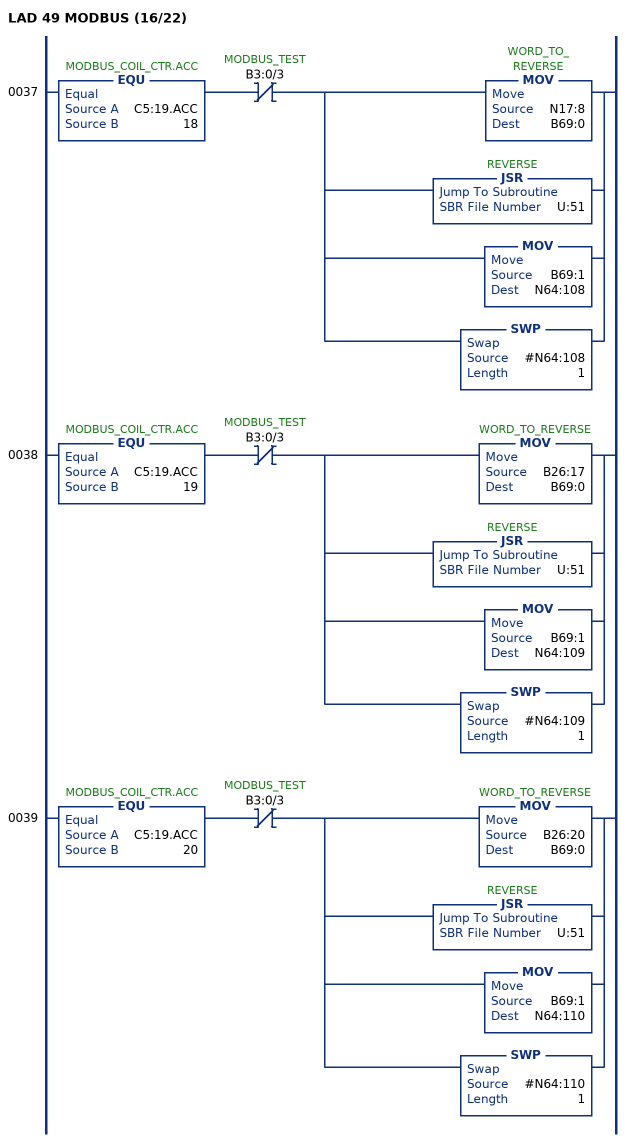
% Rung: 37 %
SOR EQU C5:19.ACC 18 XIO B3:0/3 BST MOV N17:8 B69:0 NXB JSR U:51 NXB MOV B69:1 N64:108 NXB SWP #N64:108 1 BND EOR
%   C5:19  MODBUS_COIL_CTR %
%   B3:0/3  MODBUS_TEST %
%   N17:8  ADS_B_PURIFY_WARNS  "WARNING ADS B Warnings" %
%   B69:0  WORD_TO_REVERSE %
%   U:51  REVERSE %
%   B69:1  REVERSED_WORD %
% Rung: 38 %
SOR EQU C5:19.ACC 19 XIO B3:0/3 BST MOV B26:17 B69:0 NXB JSR U:51 NXB MOV B69:1 N64:109 NXB SWP #N64:109 1 BND EOR
%   C5:19  MODBUS_COIL_CTR %
%   B3:0/3  MODBUS_TEST %
%   B26:17  GETTER_1_ALARMS %
%   B69:0  WORD_TO_REVERSE %
%   U:51  REVERSE %
%   B69:1  REVERSED_WORD %
% Rung: 39 %
SOR EQU C5:19.ACC 20 XIO B3:0/3 BST MOV B26:20 B69:0 NXB JSR U:51 NXB MOV B69:1 N64:110 NXB SWP #N64:110 1 BND EOR
%   C5:19  MODBUS_COIL_CTR %
%   B3:0/3  MODBUS_TEST %
%   B26:20  GET_1_OPEN_TC_ALARMS %
%   B69:0  WORD_TO_REVERSE %
%   U:51  REVERSE %
%   B69:1  REVERSED_WORD %

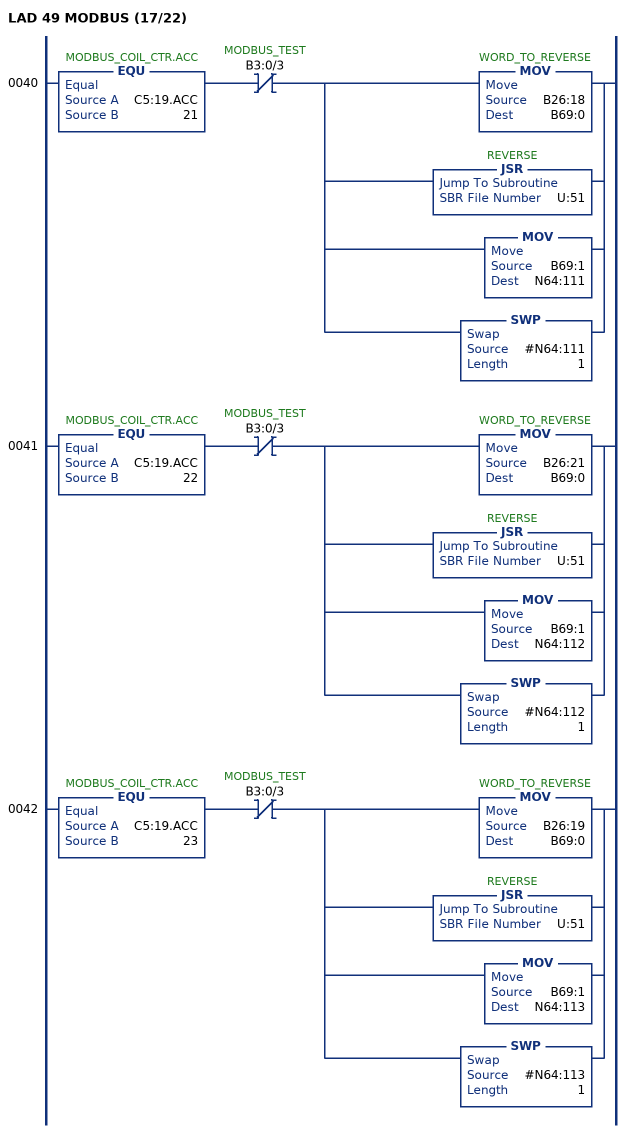
% Rung: 40 %
SOR EQU C5:19.ACC 21 XIO B3:0/3 BST MOV B26:18 B69:0 NXB JSR U:51 NXB MOV B69:1 N64:111 NXB SWP #N64:111 1 BND EOR
%   C5:19  MODBUS_COIL_CTR %
%   B3:0/3  MODBUS_TEST %
%   B26:18  GETTER_2_ALARMS %
%   B69:0  WORD_TO_REVERSE %
%   U:51  REVERSE %
%   B69:1  REVERSED_WORD %
% Rung: 41 %
SOR EQU C5:19.ACC 22 XIO B3:0/3 BST MOV B26:21 B69:0 NXB JSR U:51 NXB MOV B69:1 N64:112 NXB SWP #N64:112 1 BND EOR
%   C5:19  MODBUS_COIL_CTR %
%   B3:0/3  MODBUS_TEST %
%   B26:21  GET_2_OPEN_TC_ALARMS %
%   B69:0  WORD_TO_REVERSE %
%   U:51  REVERSE %
%   B69:1  REVERSED_WORD %
% Rung: 42 %
SOR EQU C5:19.ACC 23 XIO B3:0/3 BST MOV B26:19 B69:0 NXB JSR U:51 NXB MOV B69:1 N64:113 NXB SWP #N64:113 1 BND EOR
%   C5:19  MODBUS_COIL_CTR %
%   B3:0/3  MODBUS_TEST %
%   B26:19  GETTER_3_ALARMS %
%   B69:0  WORD_TO_REVERSE %
%   U:51  REVERSE %
%   B69:1  REVERSED_WORD %

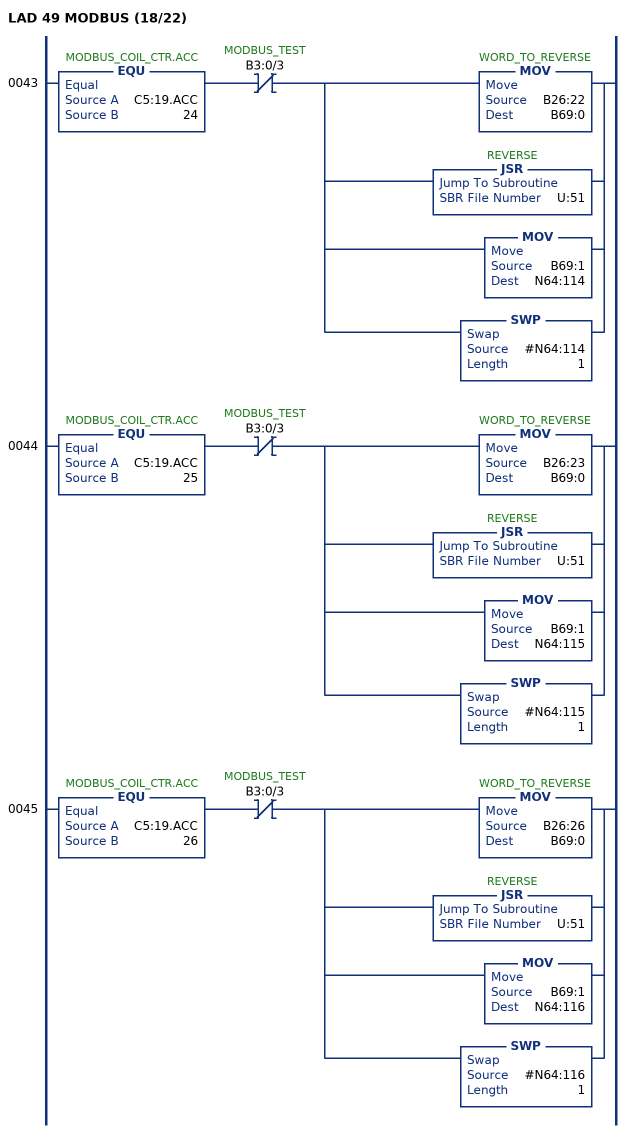
% Rung: 43 %
SOR EQU C5:19.ACC 24 XIO B3:0/3 BST MOV B26:22 B69:0 NXB JSR U:51 NXB MOV B69:1 N64:114 NXB SWP #N64:114 1 BND EOR
%   C5:19  MODBUS_COIL_CTR %
%   B3:0/3  MODBUS_TEST %
%   B26:22  GET_3_OPEN_TC_ALARMS %
%   B69:0  WORD_TO_REVERSE %
%   U:51  REVERSE %
%   B69:1  REVERSED_WORD %
% Rung: 44 %
SOR EQU C5:19.ACC 25 XIO B3:0/3 BST MOV B26:23 B69:0 NXB JSR U:51 NXB MOV B69:1 N64:115 NXB SWP #N64:115 1 BND EOR
%   C5:19  MODBUS_COIL_CTR %
%   B3:0/3  MODBUS_TEST %
%   B26:23  GETTER_1_WARNINGS %
%   B69:0  WORD_TO_REVERSE %
%   U:51  REVERSE %
%   B69:1  REVERSED_WORD %
% Rung: 45 %
SOR EQU C5:19.ACC 26 XIO B3:0/3 BST MOV B26:26 B69:0 NXB JSR U:51 NXB MOV B69:1 N64:116 NXB SWP #N64:116 1 BND EOR
%   C5:19  MODBUS_COIL_CTR %
%   B3:0/3  MODBUS_TEST %
%   B26:26  GET_1_OPEN_TC_WARNS %
%   B69:0  WORD_TO_REVERSE %
%   U:51  REVERSE %
%   B69:1  REVERSED_WORD %

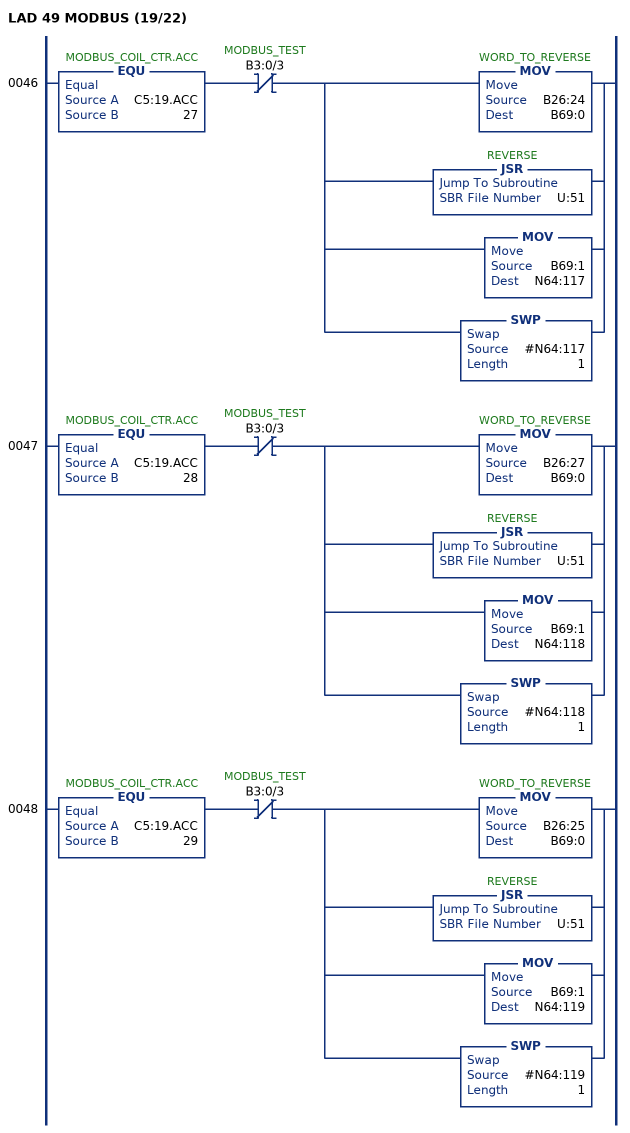
% Rung: 46 %
SOR EQU C5:19.ACC 27 XIO B3:0/3 BST MOV B26:24 B69:0 NXB JSR U:51 NXB MOV B69:1 N64:117 NXB SWP #N64:117 1 BND EOR
%   C5:19  MODBUS_COIL_CTR %
%   B3:0/3  MODBUS_TEST %
%   B26:24  GETTER_2_WARNINGS %
%   B69:0  WORD_TO_REVERSE %
%   U:51  REVERSE %
%   B69:1  REVERSED_WORD %
% Rung: 47 %
SOR EQU C5:19.ACC 28 XIO B3:0/3 BST MOV B26:27 B69:0 NXB JSR U:51 NXB MOV B69:1 N64:118 NXB SWP #N64:118 1 BND EOR
%   C5:19  MODBUS_COIL_CTR %
%   B3:0/3  MODBUS_TEST %
%   B26:27  GET_2_OPEN_TC_WARNS %
%   B69:0  WORD_TO_REVERSE %
%   U:51  REVERSE %
%   B69:1  REVERSED_WORD %
% Rung: 48 %
SOR EQU C5:19.ACC 29 XIO B3:0/3 BST MOV B26:25 B69:0 NXB JSR U:51 NXB MOV B69:1 N64:119 NXB SWP #N64:119 1 BND EOR
%   C5:19  MODBUS_COIL_CTR %
%   B3:0/3  MODBUS_TEST %
%   B26:25  GETTER_3_WARNINGS %
%   B69:0  WORD_TO_REVERSE %
%   U:51  REVERSE %
%   B69:1  REVERSED_WORD %

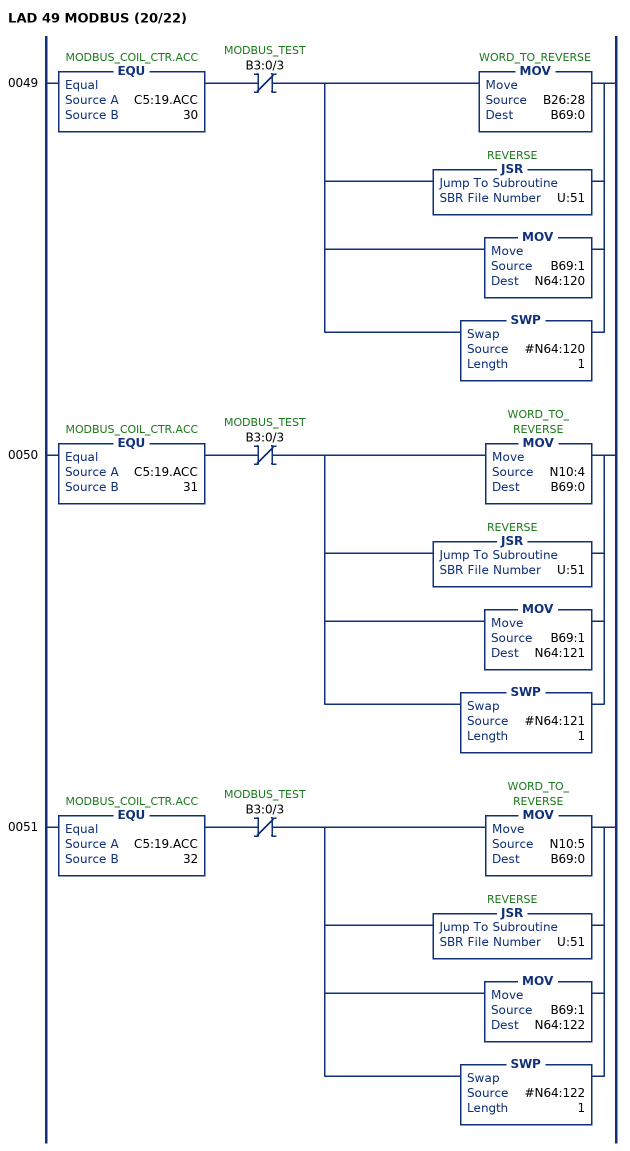
% Rung: 49 %
SOR EQU C5:19.ACC 30 XIO B3:0/3 BST MOV B26:28 B69:0 NXB JSR U:51 NXB MOV B69:1 N64:120 NXB SWP #N64:120 1 BND EOR
%   C5:19  MODBUS_COIL_CTR %
%   B3:0/3  MODBUS_TEST %
%   B26:28  GET_3_OPEN_TC_WARNS %
%   B69:0  WORD_TO_REVERSE %
%   U:51  REVERSE %
%   B69:1  REVERSED_WORD %
% Rung: 50 %
SOR EQU C5:19.ACC 31 XIO B3:0/3 BST MOV N10:4 B69:0 NXB JSR U:51 NXB MOV B69:1 N64:121 NXB SWP #N64:121 1 BND EOR
%   C5:19  MODBUS_COIL_CTR %
%   B3:0/3  MODBUS_TEST %
%   N10:4  H2_ALARMS %
%   B69:0  WORD_TO_REVERSE %
%   U:51  REVERSE %
%   B69:1  REVERSED_WORD %
% Rung: 51 %
SOR EQU C5:19.ACC 32 XIO B3:0/3 BST MOV N10:5 B69:0 NXB JSR U:51 NXB MOV B69:1 N64:122 NXB SWP #N64:122 1 BND EOR
%   C5:19  MODBUS_COIL_CTR %
%   B3:0/3  MODBUS_TEST %
%   N10:5  H2_WARNINGS %
%   B69:0  WORD_TO_REVERSE %
%   U:51  REVERSE %
%   B69:1  REVERSED_WORD %

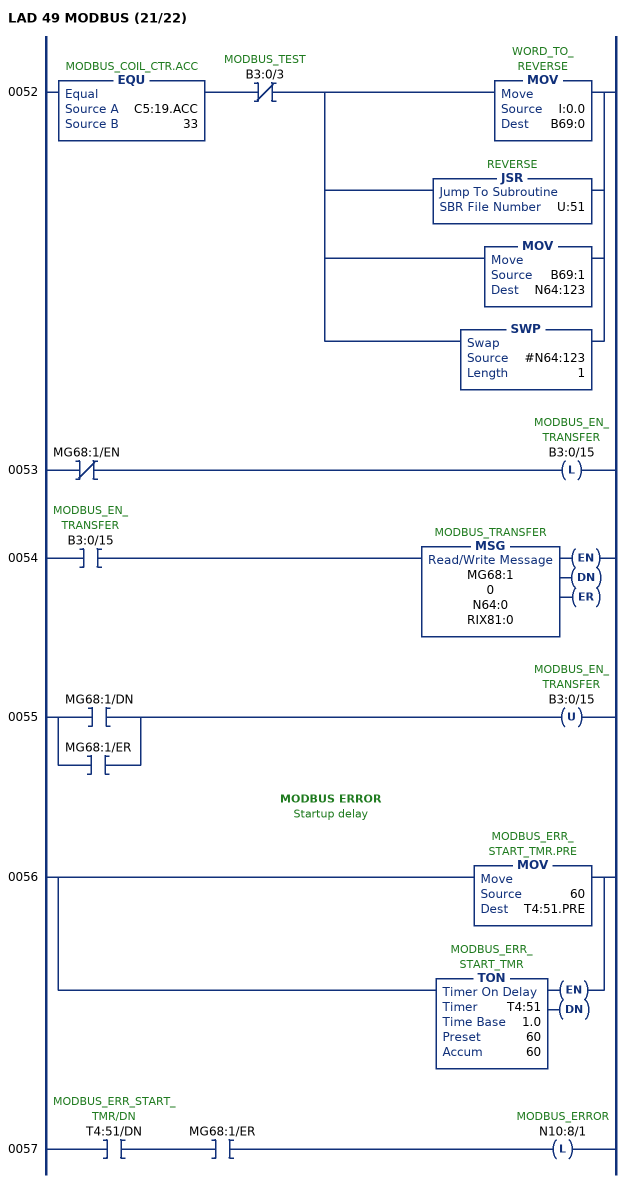
% Rung: 52 %
SOR EQU C5:19.ACC 33 XIO B3:0/3 BST MOV I:0.0 B69:0 NXB JSR U:51 NXB MOV B69:1 N64:123 NXB SWP #N64:123 1 BND EOR
%   C5:19  MODBUS_COIL_CTR %
%   B3:0/3  MODBUS_TEST %
%   B69:0  WORD_TO_REVERSE %
%   U:51  REVERSE %
%   B69:1  REVERSED_WORD %
% Rung: 53 %
SOR XIO MG68:1/EN OTL B3:0/15 EOR
%   B3:0/15  MODBUS_EN_TRANSFER %
% Rung: 54 %
SOR XIC B3:0/15 MSG MG68:1 0 N64:0 RIX81:0 EOR
%   B3:0/15  MODBUS_EN_TRANSFER %
%   MSG set-up: CIP Generic | 33 | 0 | ? | 0 | 0 | 0 | 0 | 172.16.14.73 | 0 | 0 | 172.16.14.73 | RIX81:0 | 10 | 4 | 150 | 3 | 4 | 96 | 3 | 252 | N64:0 %
%   MG68:1  MODBUS_TRANSFER %
%   N64:0  REGISTER_START %
% Rung: 55 %
SOR BST XIC MG68:1/DN NXB XIC MG68:1/ER BND OTU B3:0/15 EOR
%   B3:0/15  MODBUS_EN_TRANSFER %
% Rung: 56 %
% TITLE: MODBUS ERROR %
% Startup delay %
SOR BST MOV 60 T4:51.PRE NXB TON T4:51 1.0 60 60 BND EOR
%   T4:51  MODBUS_ERR_START_TMR %
% Rung: 57 %
SOR XIC T4:51/DN XIC MG68:1/ER OTL N10:8/1 EOR
%   T4:51  MODBUS_ERR_START_TMR %
%   N10:8/1  MODBUS_ERROR %

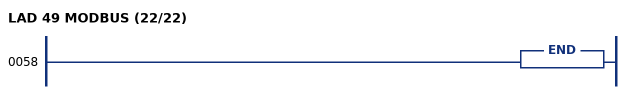
% Rung: 58 %
SOR END EOR

LADDER 50 "PLC FAULT"
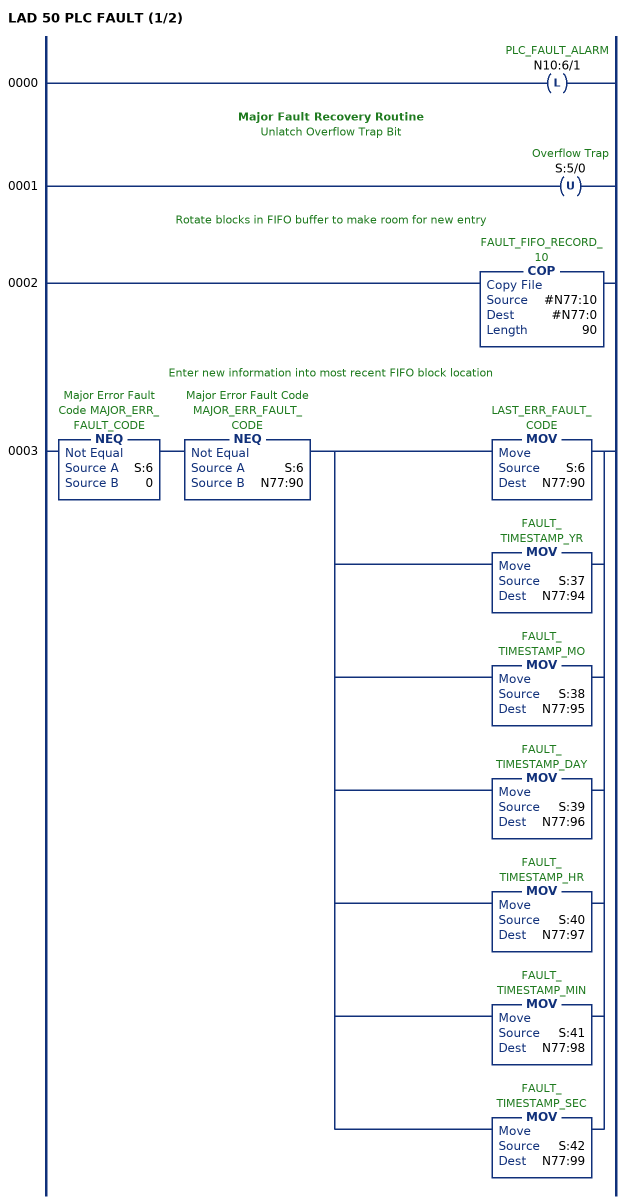
% Rung: 0 %
SOR OTL N10:6/1 EOR
%   N10:6/1  PLC_FAULT_ALARM %
% Rung: 1 %
% TITLE: Major Fault Recovery Routine %
% Unlatch Overflow Trap Bit %
SOR OTU S:5/0 EOR
%   S:5/0  "Overflow Trap" %
% Rung: 2 %
% Rotate blocks in FIFO buffer to make room for new entry %
SOR COP #N77:10 #N77:0 90 EOR
%   N77:10  FAULT_FIFO_RECORD_9 %
%   N77:0  FAULT_FIFO_RECORD_10 %
% Rung: 3 %
% Enter new information into most recent FIFO block location %
SOR NEQ S:6 0 NEQ S:6 N77:90 BST MOV S:6 N77:90 NXB MOV S:37 N77:94 NXB MOV S:38 N77:95 NXB MOV S:39 N77:96 NXB MOV S:40 N77:97 NXB MOV S:41 N77:98 NXB MOV S:42 N77:99 BND EOR
%   S:6  MAJOR_ERR_FAULT_CODE  "Major Error Fault Code" %
%   N77:90  LAST_ERR_FAULT_CODE %
%   S:37  RTC_YEAR  "Clock Calendar Year" %
%   N77:94  FAULT_TIMESTAMP_YR %
%   S:38  RTC_MONTH  "Clock Calendar Month" %
%   N77:95  FAULT_TIMESTAMP_MO %
%   S:39  RTC_DAY_OF_MONTH  "Clock Calendar Day" %
%   N77:96  FAULT_TIMESTAMP_DAY %
%   S:40  RTC_HOUR  "Clock Calendar Hours" %
%   N77:97  FAULT_TIMESTAMP_HR %
%   S:41  RTC_MINUTE  "Clock Calendar Minutes" %
%   N77:98  FAULT_TIMESTAMP_MIN %
%   S:42  RTC_SECOND  "Clock Calendar Seconds" %
%   N77:99  FAULT_TIMESTAMP_SEC %

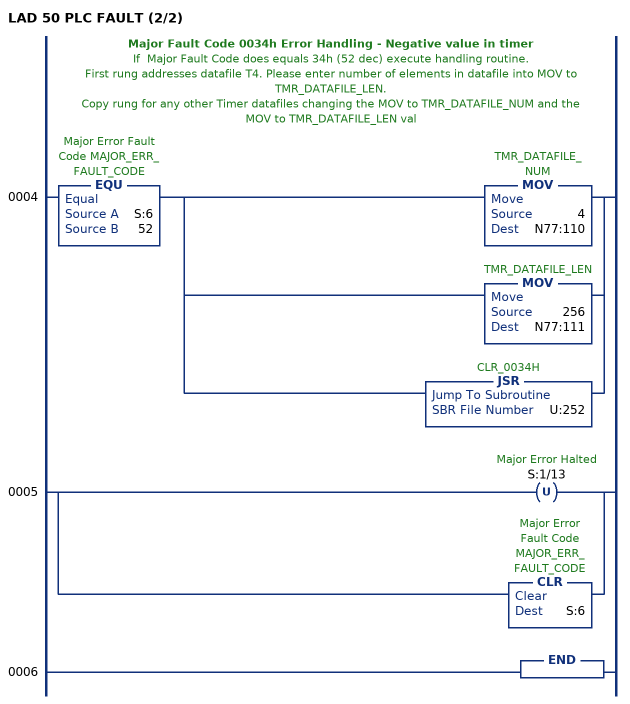
% Rung: 4 %
% TITLE: Major Fault Code 0034h Error Handling - Negative value in timer %
% If  Major Fault Code does equals 34h (52 dec) execute handling routine.
% First rung addresses datafile T4. Please enter number of elements in datafile into MOV to TMR_DATAFILE_LEN.
% Copy rung for any other Timer datafiles changing the MOV to TMR_DATAFILE_NUM and the MOV to TMR_DATAFILE_LEN val %
SOR EQU S:6 52 BST MOV 4 N77:110 NXB MOV 256 N77:111 NXB JSR U:252 BND EOR
%   S:6  MAJOR_ERR_FAULT_CODE  "Major Error Fault Code" %
%   N77:110  TMR_DATAFILE_NUM %
%   N77:111  TMR_DATAFILE_LEN %
%   U:252  CLR_0034H %
% Rung: 5 %
SOR BST OTU S:1/13 NXB CLR S:6 BND EOR
%   S:1/13  "Major Error Halted" %
%   S:6  MAJOR_ERR_FAULT_CODE  "Major Error Fault Code" %
% Rung: 6 %
SOR END EOR

LADDER 51 "REVERSE"
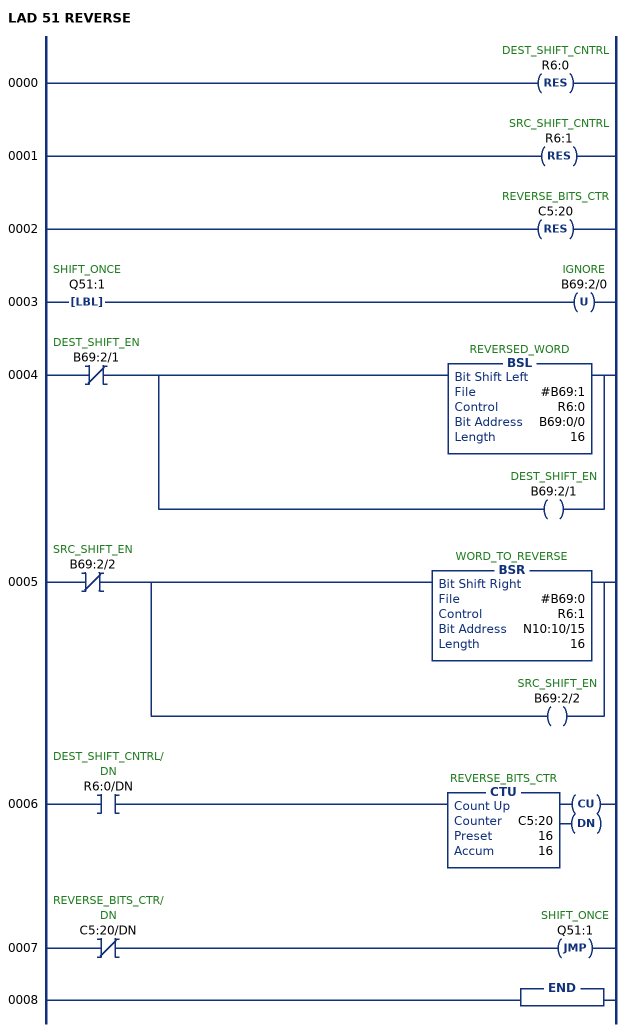
% Rung: 0 %
SOR RES R6:0 EOR
%   R6:0  DEST_SHIFT_CNTRL %
% Rung: 1 %
SOR RES R6:1 EOR
%   R6:1  SRC_SHIFT_CNTRL %
% Rung: 2 %
SOR RES C5:20 EOR
%   C5:20  REVERSE_BITS_CTR %
% Rung: 3 %
SOR LBL Q51:1 OTU B69:2/0 EOR
%   Q51:1  SHIFT_ONCE %
%   B69:2/0  IGNORE %
% Rung: 4 %
SOR XIO B69:2/1 BST BSL #B69:1 R6:0 B69:0/0 16 NXB OTE B69:2/1 BND EOR
%   B69:2/1  DEST_SHIFT_EN %
%   B69:1  REVERSED_WORD %
%   R6:0  DEST_SHIFT_CNTRL %
% Rung: 5 %
SOR XIO B69:2/2 BST BSR #B69:0 R6:1 N10:10/15 16 NXB OTE B69:2/2 BND EOR
%   B69:2/2  SRC_SHIFT_EN %
%   B69:0  WORD_TO_REVERSE %
%   R6:1  SRC_SHIFT_CNTRL %
%   N10:10/15  ALWAYS_OFF  "If this is off, go ahead and turn it off" %
% Rung: 6 %
SOR XIC R6:0/DN CTU C5:20 16 16 EOR
%   R6:0  DEST_SHIFT_CNTRL %
%   C5:20  REVERSE_BITS_CTR %
% Rung: 7 %
SOR XIO C5:20/DN JMP Q51:1 EOR
%   C5:20  REVERSE_BITS_CTR %
%   Q51:1  SHIFT_ONCE %
% Rung: 8 %
SOR END EOR

LADDER 252 "CLR_0034"
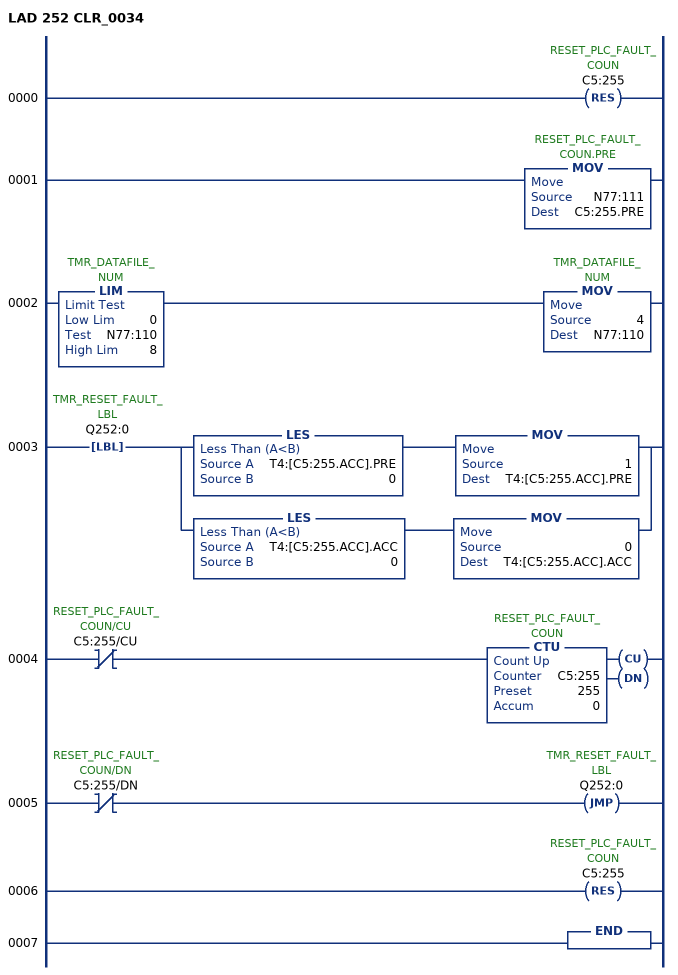
% Rung: 0 %
SOR RES C5:255 EOR
%   C5:255  RESET_PLC_FAULT_COUN %
% Rung: 1 %
SOR MOV N77:111 C5:255.PRE EOR
%   N77:111  TMR_DATAFILE_LEN %
%   C5:255  RESET_PLC_FAULT_COUN %
% Rung: 2 %
SOR LIM 0 N77:110 8 MOV 4 N77:110 EOR
%   N77:110  TMR_DATAFILE_NUM %
% Rung: 3 %
SOR LBL Q252:0 BST LES T4:[C5:255.ACC].PRE 0 MOV 1 T4:[C5:255.ACC].PRE NXB LES T4:[C5:255.ACC].ACC 0 MOV 0 T4:[C5:255.ACC].ACC BND EOR
%   Q252:0  TMR_RESET_FAULT_LBL %
%   C5:255  RESET_PLC_FAULT_COUN %
% Rung: 4 %
SOR XIO C5:255/CU CTU C5:255 255 0 EOR
%   C5:255  RESET_PLC_FAULT_COUN %
% Rung: 5 %
SOR XIO C5:255/DN JMP Q252:0 EOR
%   C5:255  RESET_PLC_FAULT_COUN %
%   Q252:0  TMR_RESET_FAULT_LBL %
% Rung: 6 %
SOR RES C5:255 EOR
%   C5:255  RESET_PLC_FAULT_COUN %
% Rung: 7 %
SOR END EOR

OTHER DOCUMENTED ADDRESSES
  B3:1/1  PLC_CLOCK_UPDATE
  B3:1/2  FIRST_SCAN_HMI
  B22:0/0  START_VENT_ADS_1_DN
  B22:0/1  START_VENT_GET_1_DN
  B22:0/2  START_HEAT_DN
  B22:0/3  START_VENT_ALL_DN
  B22:0/4  START_BKFL_1_DN
  B22:0/5  START_VENT_ADS_2_DN
  B22:0/6  START_VENT_GET_2_DN
  B22:0/7  START_BKFL_2_DN
  B26:0/1  UPS_FAIL_ALM_EN
  B26:1/5  LP_INLET_GAS_ALM_EN
  B26:5/1  UPS_FAIL_WRN_EN
  B26:6/5  LP_INLET_GAS_WRN_EN
  B26:8/1  OPEN_TC1_WARN_EN
  B26:8/2  OPEN_TC2_WARN_EN
  B26:8/3  OPEN_TC3_WARN_EN
  B26:8/4  OPEN_TC4_WARN_EN
  B26:8/6  OPEN_TC6_WARN_EN
  B26:8/7  OPEN_TC7_WARN_EN
  B26:8/8  OPEN_TC8_WARN_EN
  B26:8/9  OPEN_TC9_WARN_EN
  B26:8/11  OPEN_TC11_WARN_EN
  B26:8/12  OPEN_TC12_WARN_EN
  B26:8/13  OPEN_TC13_WARN_EN
  B26:8/14  OPEN_TC14_WARN_EN
  B26:10  GETTER_ENABLE_BITS
  B26:14/1  DIS_GET_LT_BED_FLT
  B30:0  CONFIG_BITS_HARDWARE  "CONFIG Hardware options installed"
  B30:0/7  OUTLET_PX_INSTALLED  "PX-3 Installed"
  B30:1  CONFIG_BITS_HARDWRE2  "CONFIG Hardware options installed"
  B30:1/5  THREE_GETTER_CONFIG
  B30:5  SYSTEM_STATUS_0  "STATUS System Status of system contro entities"
  B30:5/12  X_PURGE_FAIL_TO_INIT
  B31:2  SYSTEM_HMI_CMD_0  "COMMAND HMI Commands"
  B31:3  SYSTEM_HMI_CMD_1  "COMMAND HMI Commands"
  B31:3/10  DEF_LP_INLET_GAS
  B31:4  SYSTEM_HMI_CMD_2  "COMMAND HMI Commands"
  B31:5  SYSTEM_HMI_CMD_3
  B31:6  SYSTEM_HMI_CMD_4  "COMMAND HMI Commands"
  B31:7  SYSTEM_HMI_CMD_5  "COMMAND HMI Commands"
  B31:8  SYSTEM_HMI_CMD_6  "COMMAND HMI Commands"
  B33:0  PURIFY_HMI_CMDS
  B33:0/1  DEF_PURIFY_MAX
  B34:0  REGEN_HMI_CMDS
  B34:1/1  HIGH_INLET_FLW
  B34:2  REGEN_FLAGS
  B34:3  REGEN_DEF_BUTTONS
  B35:2  MANUAL_HMI_CMNDS_0
  B36:0  PURGE_DEF_BUTTONS
  B36:1  PURGE_FLAGS
  C5:8  REGEN_PURGE_MINUTES  "COUNTER Regen THe number of minutes the purge step runs"
  C5:23  X_PURGE_INIT_MIN_CTR
  DFILE:0  "OUTPUT"
  DFILE:1  "INPUT"
  DFILE:2  "STATUS"
  DFILE:3  "BINARY"
  DFILE:4  "TIMER"
  DFILE:5  "COUNTER"
  DFILE:6  "CONTROL"
  DFILE:7  "SYSTEM CFG Maintains the values that characterize t he system"
  DFILE:8  "FLOAT"
  DFILE:9  "CONSTANTS The collection of sy stem and subsystem c onstants"
  DFILE:10  "SYSTEM Contain the values f or system control"
  DFILE:11  "PROCESS Contains the values for the processing m achine"
  DFILE:12  "PURIFY Contains the values required for purify"
  DFILE:13  "REGEN Contains the values required for regen"
  DFILE:14  "PID"
  DFILE:15  "MANUAL CTL Contains the data fo r the manual valve c ontrol"
  DFILE:16  "ADSORBER_A Contains the values for Adsorber A"
  DFILE:17  "ADSORBER_B Contains the values required for Adsorbe r B"
  DFILE:18  "GETTER CMN"
  DFILE:19  "BYPASS"
  DFILE:20  "PURGE"
  DFILE:21  "STARTUP"
  DFILE:22  "STARTUP"
  DFILE:23  "GETTER 1"
  DFILE:24  "GETTER 2"
  DFILE:25  "GETTER 3"
  DFILE:26  "FAULTS"
  DFILE:27  "QUICK STRT"
  DFILE:29  "GETTER"
  DFILE:30  "SYSTEM CFG"
  DFILE:31  "SYSTEM"
  DFILE:32  "PROCESS"
  DFILE:33  "PURIFY"
  DFILE:34  "REGEN"
  DFILE:35  "MANUAL CTL"
  DFILE:36  "PURGE"
  DFILE:37  "GETTER 3"
  DFILE:38  "BYPASS"
  DFILE:51  "LONG"
  DFILE:55  "TEST_START Simultation Start"
  DFILE:60  "READ_SBC"
  DFILE:61  "WRITE_SBC"
  DFILE:64  "MODBUS"
  DFILE:68  "COMMS"
  DFILE:69  "REVERSE"
  N7:1  CONFIG_BITS_ALM_O  "CONFIG System alarms enable"
  N7:2  CONFIG_BITS_ALM_1  "CONFIG System alarms enable"
  N7:3  CONFIG_BITS_WARN_0  "CONFIG System warnings enable"
  N7:4  CONFIG_BITS_WARN_1  "CONFIG System warnings enable"
  N7:5  CALENDER_YEAR
  N7:6  CALENDER_MONTH
  N7:7  CALENDER_DAY
  N7:8  CALENDER_HOUR
  N7:9  CALENDER_MINUTE
  N7:10  CALENDER_SECOND
  N7:70  LP_INLET_GAS_ALM_SP
  N7:71  LP_INLET_GAS_WRN_SP
  N9:60  QUICK_IDLE
  N9:61  QUICK_VENT_ALL
  N9:62  QUICK_BACKFILL_1
  N9:63  QUICK_VENT
  N9:64  QUICK_BACKFILL_2
  N9:65  QUICK_BACKFILL_3
  N9:66  QUICK_COOL
  N9:67  QUICK_DONE
  N10:2  GETTER_ALARMS
  N10:3  GETTER_WARNINGS
  N10:6/14  LP_INLET_GAS_ALARM
  N10:8/14  LP_INLET_GAS_WARN
  N10:10  SYSTEM_CONTROL  "CONTROL System Bits used to manipulate hardware"
  N10:14  DIF_TRANS_PRESSURE
  N10:16  SYSTEM_FLAGS_1
  N11:2  PROC_ALARM_BUFFER  "STATE This holds the state of the process when the system alarm occured"
  N12:4  PURIFY_FLAGS_0  "STATUS Flags used by the purify process"
  N12:5  PURIFY_CONTROL  "CONTROL Control bits used by the purify process to change hardware states"
  N12:5/0  PURIFY_OPEN_IN_OUT  "CONTROL Purify Open the ADS purify in out valves"
  N12:6  PURIFY_COMPLETE  "STATUS Purify complete"
  N12:12  PURIFY_CALC_0  "CONFIG Math result placeholder for the purify time calculation"
  N12:13  PURIFY_FACTOR_TIME  "CONFIG The factored purify time accounting for the purify percent factor (hours)"
  N12:14  PURIFY_MAX_TIME
  N13:5  REGEN_CONTROL  "CONTROL Regen Bits used to manipulate hardware"
  N13:5/3  REGEN_OPEN_PROC_IN
  N13:5/8  REGEN_OPEN_EQUALIZE
  N13:6  REGEN_COMPLETE  "STATUS Regen complete"
  N13:9  BLANKET_LIMIT
  N14:0  QUICK_START_STATE
  N14:1  QUICK_STRT_STATE_BFR
  N15:4  MANUAL_FLAGS_0
  N16:3  ADS_A_FLAGS_0  "STATUS Flags used for Adsorber A"
  N17:3  ADS_B_FLAGS_0  "STATUS Flags used for Adsorber B"
  N19:1  BYPASS_COMMAND  "HMI Commands received from the HMI"
  N21:18  START_PURGE_CYCLES
  N21:24  START_VENT_ALL_PX
  N21:51/0  QUICK_START_VENT
  N21:51/1  QUICK_START_BACKFILL
  N21:70  QUICK_REG_RUN_TIME
  N21:71  QUICK_REG_BLEED_FLW
  N21:72  QUICK_REG_BKFIL_FLW
  REGEN_BKFIL_2_ENDPRS  
  REGEN_BKFL_2_ENDPRS  
  T4:92  LP_INLET_GAS_ALM_TMR
  T4:93  LP_INLET_GAS_WRN_TMR
  T4:113  X_PURGE_INIT_TMR
  T4:154  REGEN_STANDBY_DELAY
  T48:0  REGEN_EQUALIZE_SEC
  U:60  IO_CONFIG

COMMENTS NOT ATTACHED TO A CURRENT RUNG
  N7:8: Scale analog inputs / TODO: Do we need to add the ability to adjust the ammonia sensor scaling?
  N10:5/2: H2 SENSOR START UP DELAY / The H2 Sensor takes some time warm up until it can detect. The first scan triggers the H2 Sensor Start up delay until the H2 signal is on. The H2 sensor start up delay turns off at this time.
  RUNG000021-000020: End
  RUNG000023-000020: End
  RUNG000023-000019: ADS B Wall Temp Thermocouple warning
  T4:94: Startup Delay Timer
  B26:14/0: LOW TEMP GETTER BED
  B30:5/7: X Purge
  T4:55: Preheater Fail to Heat
  N7:109: DEFAULT PID SETTINGS
  N10:26: MFM / CONFIGURE MFM AND FLOW
  B34:2/3: SBC in REGEN flag
  B30:5/12: X-Purge
  B34:3/0: Start REGEN on an EXOTHERMED bed after an EXOTHERM triggered bed swap.
  N7:3/4: If the alarm is not enabled for a specified amount of time, turn it back on.
  N10:25: MASS FLOW METER

REVISION NOTES
  0: moved some bits out of N7 into B30
  1: moved bits out of N10 into B31
  2: moved bits from N15 into B35
  3: added the final data files. didn't need to move any bits
  4: updated configuration for TC and AI cards. updated DO module point assignments
  5: added logic for double-acting purify valves
  6: added rod and blanket limits
  7: added tags for default buttons
  8: cleaning up bed b pid control code
  9: removed h2 sensor and moved moisture sensor to channel 6
  10: changed processor name
  11: added px3 reading
  12: added call to mix panel routine
  13: test ok
  14: trying to clear plc fault by entering new pid default parameters
  15: changed stored PID values so that it maybe doesn't fault the PLC
  16: copid in new PID values from PS21
  17: cleared out the data table
  18: changed ADS_TC_OPEN_SP to 13700 by default
  19: setting default PID parameters
  20: added in preheater and blanket setpoints
  21: lots of changes to PID control
  22: fixed up PID defaults
  23: done testing
  24: got rid of separate PID defaults
  25: fixed loop update time bug in preheater defaults
  26: PID control done
  27: ok, now it's done. made Adsorber B use the same PID parameters as Adsorber A.
  28: added control for AV11 to system routine
  29: moved mixing panel valves into mixing panel routine
  30: some small fixes to the processing subroutine.
  31: cleaned up manual valve control for AV10, 11
  32: minor edit to purify factor calculation
  33: made some fixes to ADS_A routine including adding another state buffer for adsorber-only alarms.
  34: fixed up ADS_B routine so that it's like ADS_B
  35: Regen sequence modified and default regen paramters added
  36: added regen default comments
  37: added regen steps to constants
  38: Regen counter condition resets added
  39: Fixed regen standby buffer
  40: Regen buffering and sequencing checked and fixed
  41: Merged
  42: remove alarm aknowledge
  43: Updated alarm tag names
  44: PH fault changed
  45: manual mode PID taop PID control
  46: Added fail to cool alarm and warning
  47: trying to fix ph fault
  48: fixing open tc
  49: fixed open tc logic
  50: ok, now it's fixed

DATA TABLE (non-zero values as saved)
DATA T4
% .PRE .ACC %
% T4:0 % 6 0
% T4:1 % 60 0
% T4:2 % 6 0
% T4:3 % 100 0
% T4:4 % 60 0
% T4:5 % 60 0
% T4:6 % 1000 0
% T4:7 % 1000 0
% T4:8 % 5 0
% T4:9 % 5 0
% T4:10 % 5 0
% T4:11 % 5 0
% T4:12 % 5 0
% T4:14 % 5 0
% T4:16 % 18000 0
% T4:17 % 18000 0
% T4:18 % 18000 0
% T4:19 % 18000 0
% T4:20 % 5 0
% T4:22 % 5 0
% T4:24 % 1 0
% T4:25 % 1 0
% T4:26 % 5 0
% T4:27 % 5 0
% T4:28 % 5 0
% T4:29 % 5 0
% T4:30 % 60 0
% T4:31 % 60 0
% T4:32 % 5 0
% T4:33 % 5 0
% T4:34 % 2 0
% T4:35 % 5 0
% T4:36 % 5 0
% T4:37 % 5 0
% T4:38 % 5 0
% T4:39 % 5 0
% T4:40 % 5 0
% T4:41 % 5 0
% T4:42 % 5 0
% T4:43 % 5 0
% T4:44 % 60 0
% T4:45 % 120 0
% T4:46 % 60 0
% T4:47 % 120 0
% T4:48 % 60 0
% T4:49 % 60 0
% T4:50 % 60 0
% T4:51 % 60 60
% T4:52 % 2 0
% T4:53 % 2 0
% T4:54 % 60 0
% T4:55 % 60 0
% T4:56 % 2 0
% T4:57 % 2 0
% T4:58 % 2 0
% T4:59 % 2 0
% T4:60 % 5 0
% T4:61 % 5 0
% T4:62 % 5 0
% T4:63 % 5 5
% T4:64 % 5 0
% T4:65 % 5 5
% T4:66 % 5 0
% T4:67 % 5 0
% T4:68 % 5 0
% T4:69 % 5 0
% T4:70 % 5 0
% T4:71 % 5 0
% T4:72 % 5 0
% T4:73 % 5 0
% T4:74 % 60 0
% T4:75 % 60 0
% T4:76 % 60 0
% T4:77 % 60 0
% T4:78 % 5 0
% T4:79 % 5 0
% T4:80 % 5 0
% T4:81 % 5 0
% T4:82 % 5 0
% T4:84 % 5 0
% T4:86 % 5 0
% T4:88 % 5 0
% T4:90 % 600 0
% T4:91 % 600 0
% T4:92 % 5 0
% T4:93 % 5 0
% T4:94 % 2 0
% T4:95 % 2 0
% T4:96 % 5 0
% T4:97 % 5 0
% T4:98 % 5 0
% T4:99 % 5 0
% T4:100 % 5 0
% T4:101 % 5 0
% T4:102 % 5 5
% T4:103 % 5 0
% T4:104 % 60 0
% T4:105 % 60 0
% T4:106 % 15 0
% T4:107 % 30 0
% T4:108 % 5 0
% T4:110 % 5 0
% T4:112 % 5 0
% T4:113 % 60 0
% T4:114 % 900 0
% T4:115 % 900 0
% T4:116 % 1000 0
% T4:117 % 1000 0
% T4:118 % 1000 0
% T4:119 % 1000 0
% T4:120 % 5 0
% T4:122 % 5 0
% T4:124 % 5 0
% T4:126 % 5 0
% T4:128 % 5 0
% T4:129 % 5 0
% T4:130 % 5 0
% T4:131 % 5 0
% T4:132 % 5 0
% T4:133 % 5 0
% T4:135 % 5 0
% T4:136 % 5 0
% T4:137 % 5 0
% T4:138 % 5 0
% T4:139 % 5 0
% T4:140 % 5 0
% T4:141 % 5 0
% T4:142 % 5 0
% T4:143 % 5 0
% T4:144 % 5 0
% T4:145 % 5 0
% T4:146 % 5 0
% T4:147 % 5 0
% T4:148 % 5 0
% T4:149 % 5 0
% T4:150 % 10 0
% T4:151 % 1000 58
% T4:152 % 100 0
% T4:153 % 100 73
% T4:154 % 1 0
% T4:155 % 2 2
% T4:156 % 60 19
% T4:157 % 2 0
% T4:159 % 900 0
% T4:160 % 1000 0
% T4:161 % 1000 0
% T4:162 % 5 0
% T4:164 % 5 0
% T4:166 % 5 0
% T4:168 % 5 0
% T4:170 % 500 0
% T4:171 % 180 180
% T4:172 % 2 2
DATA C5
% .PRE .ACC %
% C5:0 % 168 0
% C5:1 % 60 0
% C5:2 % 24 0
% C5:3 % 32767 0
% C5:4 % 480 0
% C5:5 % 180 0
% C5:6 % 4 0
% C5:7 % 8 0
% C5:8 % 480 0
% C5:9 % 30 0
% C5:10 % 30 0
% C5:11 % 30 0
% C5:12 % 600 0
% C5:13 % 600 0
% C5:14 % 8 0
% C5:15 % 10 0
% C5:16 % 32767 0
% C5:17 % 480 0
% C5:18 % 480 0
% C5:19 % 34 2
% C5:20 % 16 16
% C5:21 % 30 0
% C5:22 % 30 0
% C5:255 % 255 0
DATA R6
% .LEN .POS %
% R6:0 % 16 0
% R6:1 % 16 0
DATA T252
% .PRE .ACC %
% T252:0 % 60 0
% T252:1 % 60 0
% T252:2 % 60 0
% T252:3 % 60 0
% T252:4 % 60 0
DATA C253
% .PRE .ACC %
% C253:0 % 10 0
% C253:1 % 10 0
% C253:2 % 10 0
% C253:3 % 10 0
% C253:4 % 10 0
% C253:5 % 10 0
